TYPE E_Subsystem :
(
	VACUUM := 'VACUUM',
	MPS := 'MPS',
	MOTION := 'MOTION',
	FIELDBUS := 'FIELDBUS',
	NILVALUE := '-'
)STRING;
END_TYPE

(* stored: Version 1.1.0.1, ProductVersion 3.1.4018.5
   DUT E_Subsystem: Id {0625d196-cb6d-4bee-9ee7-7900621abd78} *)
